(* CODESYS project Industrial_Tank_Control.export

Project tree, tasks and I/O mapping:
  Device : CODESYS Control Win V3 x64, CODESYS, version 3.5.22.30
    application Application
      libraries: Standard, 3.5.22.0 (System)
      task AlarmManagerTask (cyclic, interval 50 ms, priority 31) calls AlarmManager.Alarm_Prg
      task MainTask (cyclic, interval t#20ms, priority 1) calls PRG_LevelInputProcessing, PLC_PRG, PRG_TankSimulation
      task VISU_TASK (cyclic, interval 100 ms, priority 31) calls VisuElems.Visu_Prg
      Alarm Configuration
        alarm class Error (priority 10, acknowledge ACK_REP)
        alarm class Info (priority 100, acknowledge REP)
        alarm class Warning (priority 30, acknowledge REP)
        alarm group AG_Process
            2 [Error]: Comparison Equal, ExpressionToCompare TRUE, Expression PLC_PRG.xFaultLatched - "P-101 Motor Start Failure / Fault Latched"
            3 [Warning]: Comparison Equal, ExpressionToCompare FALSE, Expression GVL_IO.xMotorHealthy - "P-101 Motor Protection Not Healthy"
            1 [Error]: Comparison Equal, ExpressionToCompare TRUE, Expression GVL_Tank.xLevelSignalFault - "LT-101 Level Transmitter Signal Invalid | Signal at trigger: <LATCH1> mA"
            4 [Error]: Comparison Equal, ExpressionToCompare TRUE, Expression GVL_Tank.xHighHighLevelAlarm - "T-101 High-High Level >= 90% | Level at trigger: <LATCH1> %"
        AlarmStorage
        text list AG_Process
      global variables GVL_IO
      global variables GVL_Tank
      program PLC_PRG [LD]
      program PRG_LevelInputProcessing [ST]
      program PRG_TankSimulation [ST]
      visualisation VIS_EngineeringDiagnostics
      visualisation VIS_TankOverview
*)

// Device/Application/GVL_IO
VAR_GLOBAL

    // Simulated motor status signals

    xMotorFeedback : BOOL := FALSE;

    xMotorHealthy : BOOL := TRUE;


    // Simulation fault injection

    xSimulateMotorFailure : BOOL := FALSE;
	
	// Level transmitter fault injection

	xSimulateLevelSignalLoss : BOOL := FALSE;
	

END_VAR

// Device/Application/GVL_Tank
VAR_GLOBAL

    // Actual physical tank level in simulation

    rActualTankLevel : REAL := 50.0;


    // Simulated level transmitter current

    rLevelCurrent_mA : REAL := 12.0;


    // Measured tank level calculated by PLC

    rTankLevel : REAL := 50.0;


    // Level measurement validity

    xLevelSensorValid : BOOL := FALSE;
	
	
	// Level signal validity
	
	xLevelSignalFault : BOOL := FALSE;
	xHighHighLevelAlarm : BOOL := FALSE;

END_VAR

// Device/Application/PRG_LevelInputProcessing
PROGRAM PRG_LevelInputProcessing
VAR
END_VAR

// ==========================================
// ANALOG INPUT PROCESSING - LT-101
// ==========================================


// 1. Validate transmitter signal

GVL_Tank.xLevelSensorValid :=
    (GVL_Tank.rLevelCurrent_mA >= 4.0)
    AND
    (GVL_Tank.rLevelCurrent_mA <= 20.0);


// 2. Diagnostic signal fault

GVL_Tank.xLevelSignalFault :=
    NOT GVL_Tank.xLevelSensorValid;


// 3. Scale valid 4-20 mA signal to 0-100 %

IF GVL_Tank.xLevelSensorValid THEN

    GVL_Tank.rTankLevel :=
        ((GVL_Tank.rLevelCurrent_mA - 4.0) / 16.0) * 100.0;

END_IF;


// 4. High-High process alarm
// This MUST execute every PLC scan

GVL_Tank.xHighHighLevelAlarm :=
    GVL_Tank.xLevelSensorValid
    AND
    (GVL_Tank.rTankLevel >= 90.0);

END_PROGRAM

// Device/Application/PLC_PRG
PROGRAM PLC_PRG
VAR
    xStart : BOOL;
    xStop : BOOL;

    xLevelOK : BOOL;

    xRunRequest : BOOL;
    xMotorRun : BOOL;
	

    fbStartDelay : TON;
	fbFeedbackTimer : TON;
	
	tElapsedTime : TIME;
	tFeedbackWait : TIME;

	xStartFailure : BOOL;
	xFaultLatched : BOOL;
	
	xReset : BOOL;
	xResetAllowed : BOOL;
	
	fbFaultLatch : SR;
	
	fbStartEdge : R_TRIG;
	
	xStartPulse : BOOL;
	
	
	// AUTOMATIC TANK FILLING
	xFillStartCondition : BOOL;

	xFillStopCondition : BOOL;

	xInletValveCmd : BOOL;

	fbFillLatch : SR;
	
END_VAR

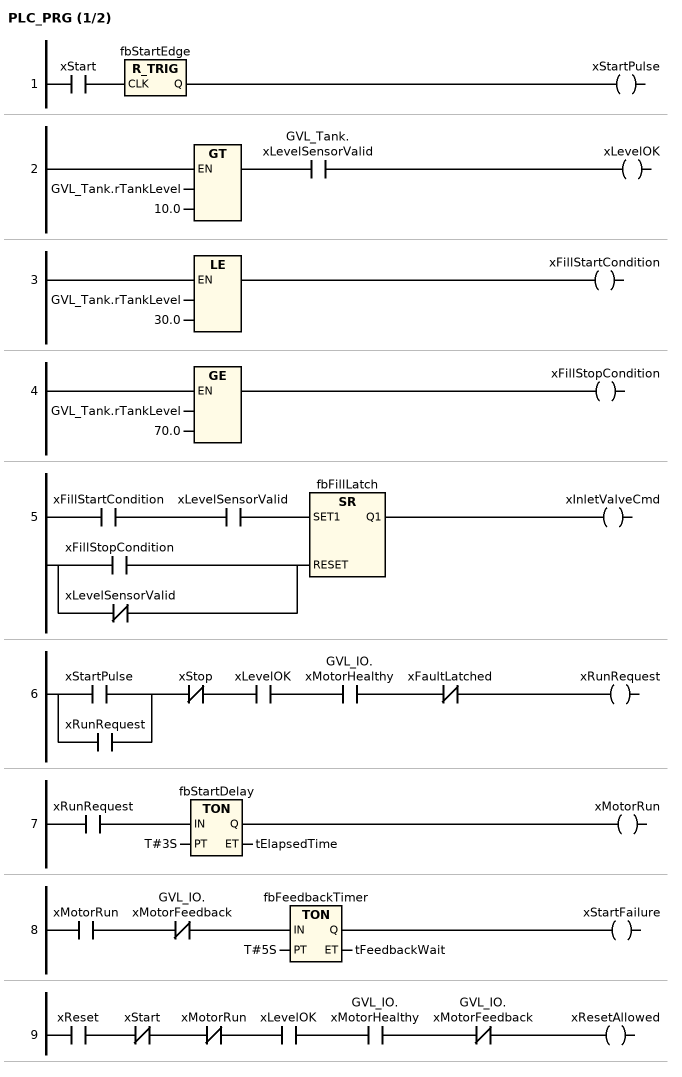
// NETWORK 1
fbStartEdge(CLK := xStart); // R_TRIG
xStartPulse := fbStartEdge.Q;

// NETWORK 2
xLevelOK := GVL_Tank.rTankLevel > 10.0 AND GVL_Tank.xLevelSensorValid;

// NETWORK 3
xFillStartCondition := GVL_Tank.rTankLevel <= 30.0;

// NETWORK 4
xFillStopCondition := GVL_Tank.rTankLevel >= 70.0;

// NETWORK 5
fbFillLatch(SET1 := xFillStartCondition AND xLevelSensorValid, RESET := xFillStopCondition OR NOT xLevelSensorValid); // SR
xInletValveCmd := fbFillLatch.Q1;

// NETWORK 6
xRunRequest := (xStartPulse OR xRunRequest) AND NOT xStop AND xLevelOK AND GVL_IO.xMotorHealthy AND NOT xFaultLatched;

// NETWORK 7
fbStartDelay(IN := xRunRequest, PT := T#3S, ET => tElapsedTime); // TON
xMotorRun := fbStartDelay.Q;

// NETWORK 8
fbFeedbackTimer(IN := xMotorRun AND NOT GVL_IO.xMotorFeedback, PT := T#5S, ET => tFeedbackWait); // TON
xStartFailure := fbFeedbackTimer.Q;

// NETWORK 9
xResetAllowed := xReset AND NOT xStart AND NOT xMotorRun AND xLevelOK AND GVL_IO.xMotorHealthy AND NOT GVL_IO.xMotorFeedback;

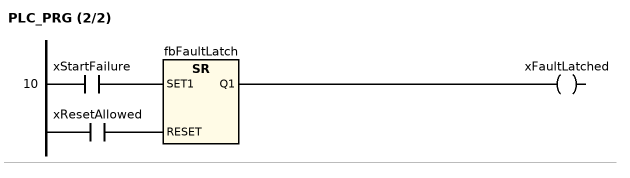
// NETWORK 10
fbFaultLatch(SET1 := xStartFailure, RESET := xResetAllowed); // SR
xFaultLatched := fbFaultLatch.Q1;

END_PROGRAM

// Device/Application/PRG_TankSimulation
PROGRAM PRG_TankSimulation
VAR

    fbPlantTick : TON;
	
	fbMotorStartSim : TON;

    rInletRatePctPerS : REAL := 2.0;

    rOutletRatePctPerS : REAL := 1.0;

END_VAR

// ==========================================
// INDUSTRIAL TANK - PROCESS SIMULATION
// ==========================================


// Generate one process update approximately every second

fbPlantTick(
    IN := NOT fbPlantTick.Q,
    PT := T#1s
);


// ==========================================
// TANK LEVEL SIMULATION
// ==========================================

IF fbPlantTick.Q THEN

    // Water entering the tank
    IF PLC_PRG.xInletValveCmd THEN

        GVL_Tank.rActualTankLevel :=
            GVL_Tank.rActualTankLevel + rInletRatePctPerS;

    END_IF;


    // Water leaving the tank
    IF PLC_PRG.xMotorRun AND GVL_IO.xMotorFeedback THEN

        GVL_Tank.rActualTankLevel :=
            GVL_Tank.rActualTankLevel - rOutletRatePctPerS;

    END_IF;


    // Keep physical level between 0 and 100 %
    IF GVL_Tank.rActualTankLevel > 100.0 THEN

        GVL_Tank.rActualTankLevel := 100.0;

    ELSIF GVL_Tank.rActualTankLevel < 0.0 THEN

        GVL_Tank.rActualTankLevel := 0.0;

    END_IF;

END_IF;


// ==========================================
// AUTOMATIC MOTOR FEEDBACK SIMULATION
// ==========================================

fbMotorStartSim(
    IN := PLC_PRG.xMotorRun
          AND GVL_IO.xMotorHealthy
          AND NOT GVL_IO.xSimulateMotorFailure,
    PT := T#2s
);


// Simulated running feedback
GVL_IO.xMotorFeedback := fbMotorStartSim.Q;


// ==========================================
// LEVEL TRANSMITTER SIMULATION - LT-101
// ==========================================

IF GVL_IO.xSimulateLevelSignalLoss THEN

    // Fault injection: transmitter signal lost
    GVL_Tank.rLevelCurrent_mA := 0.0;

ELSE

    // Normal operation:
    // 0...100 % physical level -> 4...20 mA
    GVL_Tank.rLevelCurrent_mA :=
        4.0 + (GVL_Tank.rActualTankLevel / 100.0) * 16.0;

END_IF;

END_PROGRAM

// Device/Application/VIS_EngineeringDiagnostics
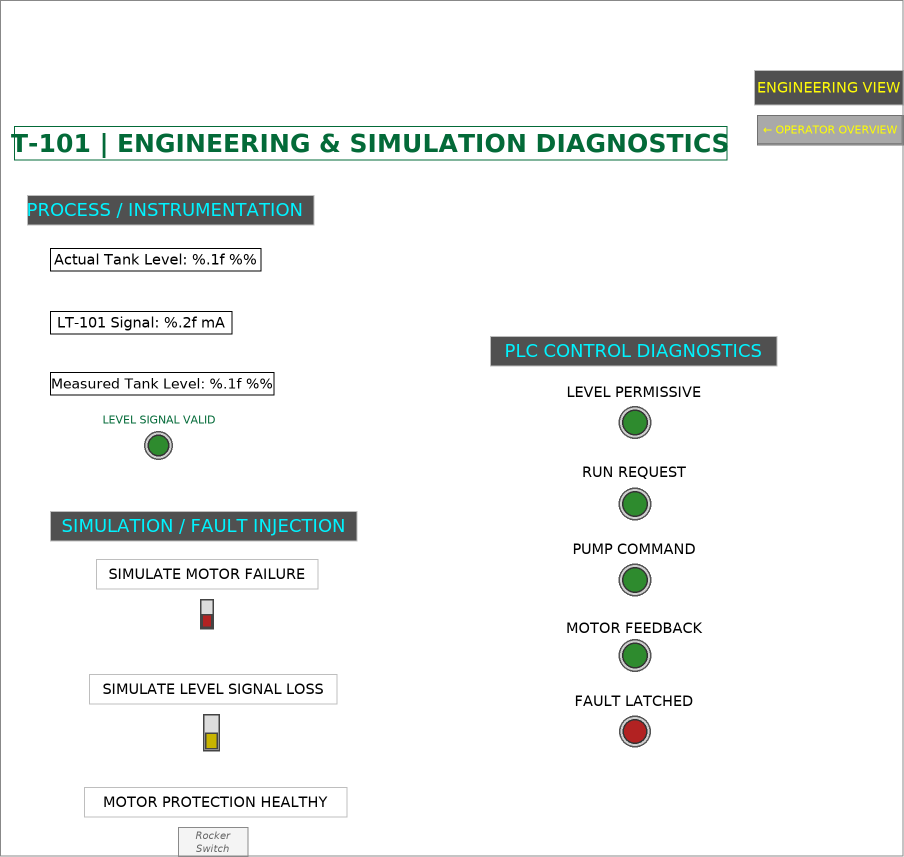
VISUALIZATION VIS_EngineeringDiagnostics  // 904x857
    Textfield (14,126 713x34), "T-101 | ENGINEERING & SIMULATION DIAGNOSTICS"
    Textfield (754,70 150x35), "ENGINEERING VIEW"
    Textfield (27,195 287x30), "PROCESS / INSTRUMENTATION"
    Textfield (490,336 287x30), "PLC CONTROL DIAGNOSTICS"
    Textfield (50,511 307x30), "SIMULATION / FAULT INJECTION"
    Textfield (50,248 211x23), "Actual Tank Level: %.1f %%", text variable: GVL_Tank.rActualTankLevel
    Textfield (50,311 182x23), "LT-101 Signal: %.2f mA", text variable: GVL_Tank.rLevelCurrent_mA
    Textfield (50,372 224x23), "Measured Tank Level: %.1f %%", text variable: GVL_Tank.rTankLevel
    Lamp1 (140,429 37x33), variable: GVL_Tank.xLevelSensorValid, style: Lamp-Lamp1-Green
    Label (98,405 122x30), "LEVEL SIGNAL VALID"
    Lamp1 (616,403 38x39), variable: PLC_PRG.xLevelOK, style: Lamp-Lamp1-Green
    Label (563,377 142x30), "LEVEL PERMISSIVE"
    Lamp1 (616,484 38x40), variable: PLC_PRG.xRunRequest, style: Lamp-Lamp1-Green
    Label (563,457 142x30), "RUN REQUEST"
    Lamp1 (616,560 38x40), variable: PLC_PRG.xMotorRun, style: Lamp-Lamp1-Green
    Label (563,534 142x30), "PUMP COMMAND"
    Lamp1 (616,635 38x41), variable: GVL_IO.xMotorFeedback, style: Lamp-Lamp1-Green
    Label (563,613 142x30), "MOTOR FEEDBACK"
    Lamp1 (616,713 38x37), variable: PLC_PRG.xFaultLatched, style: Lamp-Lamp1-Red
    Label (563,686 142x30), "FAULT LATCHED"
    DipSwitch (172,599 70x30), variable: GVL_IO.xSimulateMotorFailure, behaviour: TOGGLE, style: Switch-DipSwitch-Red
    Textfield (96,559 222x30), "SIMULATE MOTOR FAILURE"
    DipSwitch (175,714 73x37), variable: GVL_IO.xSimulateLevelSignalLoss, behaviour: TOGGLE, style: Switch-DipSwitch-Yellow
    Textfield (89,674 248x30), "SIMULATE LEVEL SIGNAL LOSS"
    RockerSwitch (178,827 70x30), variable: GVL_IO.xMotorHealthy, behaviour: TOGGLE, style: Switch-RockerSwitch-Green
    Textfield (84,787 263x30), "MOTOR PROTECTION HEALTHY"
    Button (757,115 147x30), "← OPERATOR OVERVIEW"
        OnMouseClick:  Assign=VIS_TankOverview, Type=Assignment
END_VISUALIZATION

// Device/Application/VIS_TankOverview
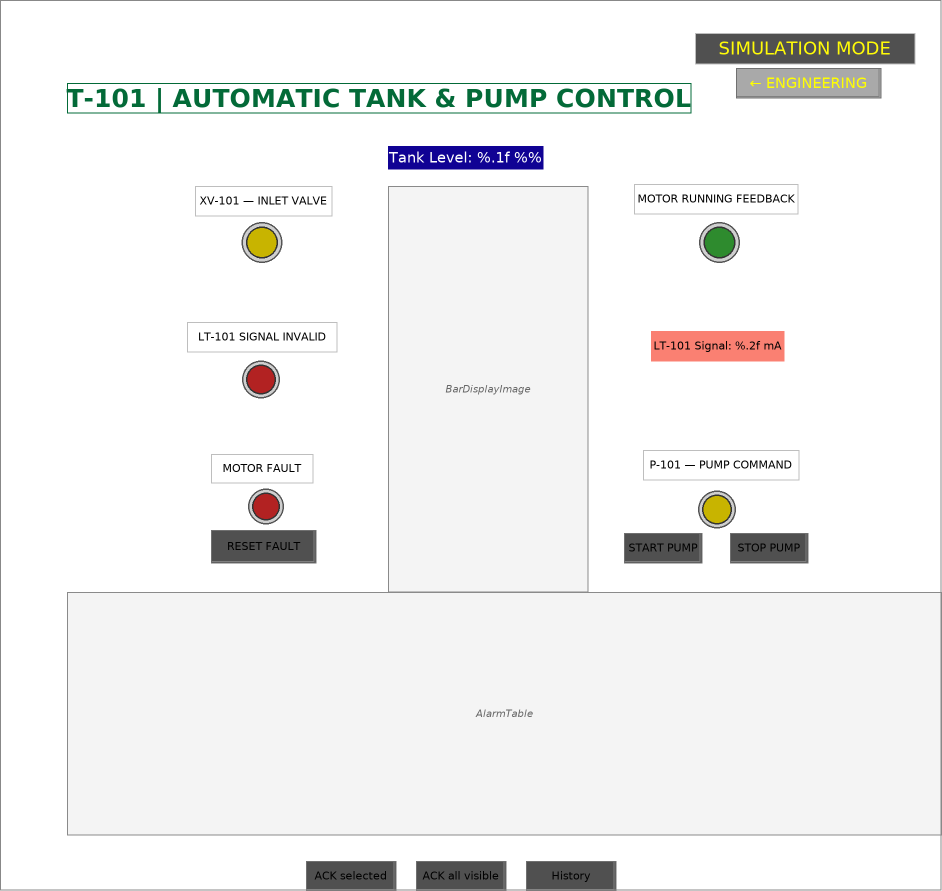
VISUALIZATION VIS_TankOverview  // 942x891
VAR_IN_OUT
END_VAR
VAR
	bAckSel : BOOL;
	bAckVisible : BOOL;
	bHistory : BOOL;
END_VAR
    BarDisplayImage (388,186 200x406), value: GVL_Tank.rTankLevel, style: BarDisplayImage-Gray, scale format: %.1f, scale 0..100
    Textfield (388,146 155x23), "Tank Level: %.1f %%", text variable: GVL_Tank.rTankLevel
    Lamp1 (238,219 48x47), variable: PLC_PRG.xInletValveCmd, style: Lamp-Lamp1-Yellow
    Lamp1 (695,485 44x49), variable: PLC_PRG.xMotorRun, style: Lamp-Lamp1-Yellow
    Textfield (195,186 137x30), "XV-101 — INLET VALVE"
    Textfield (643,450 156x30), "P-101 — PUMP COMMAND"
    Button (624,533 78x30), "START PUMP"
        tap PLC_PRG.xStart
    Button (730,533 78x30), "STOP PUMP"
        tap PLC_PRG.xStop
    Button (211,530 105x33), "RESET FAULT"
        tap PLC_PRG.xReset
    Lamp1 (242,486 48x41), variable: PLC_PRG.xFaultLatched, style: Lamp-Lamp1-Red
    Textfield (211,454 102x29), "MOTOR FAULT"
    Lamp1 (695,219 49x47), variable: GVL_IO.xMotorFeedback, style: Lamp-Lamp1-Green
    Textfield (634,184 164x30), "MOTOR RUNNING FEEDBACK"
    Textfield (695,33 220x31), "SIMULATION MODE"
    Textfield (651,331 133x30), "LT-101 Signal: %.2f mA", text variable: GVL_Tank.rLevelCurrent_mA
    Textfield (187,322 150x30), "LT-101 SIGNAL INVALID"
    Lamp1 (239,355 44x49), variable: GVL_Tank.xLevelSignalFault, style: Lamp-Lamp1-Red
    AlarmTable (67,592 875x243)
        Column[5]: ColumnTitle=Trigger Value
        p1521930926: AG_Process
        p1663851261: __All
        p428520879: bAckSel
        p2607059081: bAckVisible
        p3266827225: bHistory
    Button (306,861 90x30), "ACK selected"
        toggle bAckSel
    Button (416,861 90x30), "ACK all visible"
        toggle bAckVisible
    Button (526,861 90x30), "History"
        toggle bHistory
    Textfield (67,83 624x30), "T-101 | AUTOMATIC TANK & PUMP CONTROL"
    Button (736,68 145x30), "← ENGINEERING"
        OnMouseClick:  Assign=VIS_EngineeringDiagnostics, Type=Assignment
END_VISUALIZATION

(* text list AG_Process (id | default)
  4 | T-101 High-High Level >= 90% | Level at trigger: <LATCH1> %
  3 | P-101 Motor Protection Not Healthy
  2 | P-101 Motor Start Failure / Fault Latched
  1 | LT-101 Level Transmitter Signal Invalid | Signal at trigger: <LATCH1> mA
  0 | 
   |  *)
